INTERFACE I_AxisCommand EXTENDS I_Command

END_INTERFACE

(* stored: Version 1.1.0.1, ProductVersion 3.1.4024.12
   Itf I_AxisCommand: Id {37460c4f-fea6-4068-8c06-595679d4a379} *)
